// TIA Portal project "s14_code" (V21)

(* hardware
DEVICE "S7-1500/ET200MP station_1"  S7-1500 station
   slot 0: "Rail_0"  Rack  6ES7 590-1***0-0AA0
   slot 1: "ZZPLC"  CPU 1511-1 PN  6ES7 511-1AK00-0AB0  V1.8
      slot 3: "CPU display_1"  6ES7591-1AA00-0AA0
      slot 32768: "PROFINET interface_1"  X1
         slot 32769: "Port_1"  X1 P1
         slot 32770: "Port_2"  X1 P2
*)

// ===== PLC "ZZPLC"  CPU 1511-1 PN =====
// protected blocks, not shown: "ZZSCL"

VAR_GLOBAL   // PLC tag table "Default tag table"
   "ZZALPHA" AT %M10.0 : Bool;
   "ZZB" AT %M10.1 : Bool;
   "ZZC" AT %M10.2 : Bool;
   "ZZOUT" AT %M11.0 : Bool;
   "ZZN1" AT %MW20 : Int;
   "ZZN2" AT %MW22 : Int;
   "ZZN3" AT %MW24 : Int;
END_VAR

DATA_BLOCK "ZZDATA"   // DB1
{ S7_Optimized_Access := 'TRUE' }
VERSION : 0.1
   VAR
      run : Bool;
      speed : Int;
   END_VAR
BEGIN
END_DATA_BLOCK

DATA_BLOCK "ZZFB_DB"   // DB3
{ S7_Optimized_Access := 'TRUE' }
VERSION : 0.1
// stored: InstanceOfName ZZFB
"ZZFB"
BEGIN
END_DATA_BLOCK

DATA_BLOCK "ZZOUTER_DB"   // DB4
{ S7_Optimized_Access := 'TRUE' }
VERSION : 0.1
// stored: InstanceOfName ZZOUTER
"ZZOUTER"
BEGIN
END_DATA_BLOCK

DATA_BLOCK "ZZLAD2_DB"   // DB5
{ S7_Optimized_Access := 'TRUE' }
VERSION : 0.1
// stored: InstanceOfName ZZLAD2
"ZZLAD2"
BEGIN
END_DATA_BLOCK

// folder: System blocks/Program resources

DATA_BLOCK "IEC_Timer_0_DB"   // DB2
{ S7_Optimized_Access := 'TRUE' }
AUTHOR : Simatic
FAMILY : IEC
NAME : IEC_TMR
VERSION : 1.0
// stored: InstanceOfName IEC_TIMER
"IEC_TIMER"
BEGIN
END_DATA_BLOCK

// folder: (top level)

FUNCTION_BLOCK "ZZFB"   // FB1, LAD
{ S7_Optimized_Access := 'TRUE' }
VERSION : 0.1
   VAR_INPUT
      in1 : Bool;
   END_VAR
   VAR_OUTPUT
      out1 : Bool;
   END_VAR
   VAR_IN_OUT
      io1 : Int;
   END_VAR
BEGIN

REGION Network 1
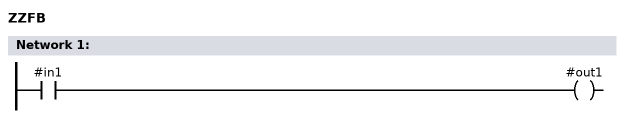
   RUNG wire#powerrail
      Contact( #in1 )
      Coil( #out1 )
   END_RUNG
   // the same network as SCL:
   #out1 := #in1;
END_REGION
END_FUNCTION_BLOCK

FUNCTION_BLOCK "ZZOUTER"   // FB2, LAD
{ S7_Optimized_Access := 'TRUE' }
VERSION : 0.1
   VAR
      inner : "ZZFB";
   END_VAR
BEGIN

REGION Network 1
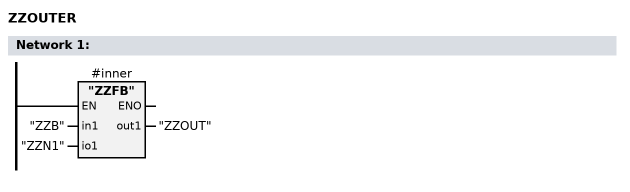
   RUNG wire#powerrail
      #inner(in1 := "ZZB", io1 := "ZZN1", out1 => "ZZOUT")
   END_RUNG
   // the same network as SCL:
   #inner(in1 := "ZZB", io1 := "ZZN1", out1 => "ZZOUT");   // "ZZFB"
END_REGION
END_FUNCTION_BLOCK

FUNCTION_BLOCK "ZZLAD2"   // FB3, LAD
{ S7_Optimized_Access := 'TRUE' }
VERSION : 0.1
   VAR
      memP : Bool;
      memN : Bool;
   END_VAR
   VAR RETAIN
      IEC_Counter_0_Instance : CTU_INT;
   END_VAR
   VAR
      IEC_Timer_0_Instance : TON_TIME;
   END_VAR
   VAR_TEMP   // added for the SCL form of the ladder/FBD networks
      _w1 : Bool;
   END_VAR
BEGIN

REGION Network 1
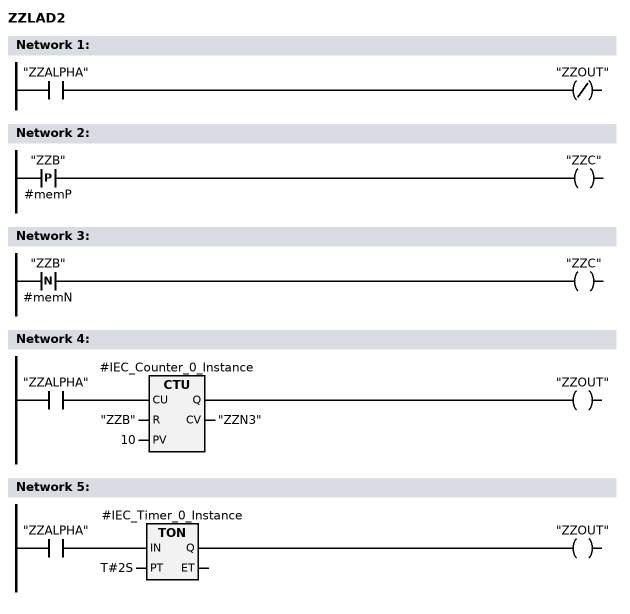
   RUNG wire#powerrail
      Contact( "ZZALPHA" )
      I_Coil( "ZZOUT" )
   END_RUNG
   // the same network as SCL:
   "ZZOUT" := NOT "ZZALPHA";
END_REGION

REGION Network 2
   RUNG wire#powerrail
      P_Contact(operand := "ZZB", bit := #memP)
      Coil( "ZZC" )
   END_RUNG
   // the same network as SCL:
   #_w1 := "ZZB" AND NOT #memP;   // rising edge of "ZZB"
   #memP := "ZZB";
   "ZZC" := #_w1;
END_REGION

REGION Network 3
   RUNG wire#powerrail
      N_Contact(operand := "ZZB", bit := #memN)
      Coil( "ZZC" )
   END_RUNG
   // the same network as SCL:
   #_w1 := NOT "ZZB" AND #memN;   // falling edge of "ZZB"
   #memN := "ZZB";
   "ZZC" := #_w1;
END_REGION

REGION Network 4
   #IEC_Counter_0_Instance(CU := "ZZALPHA", R := "ZZB", PV := 10, CV => "ZZN3");   // CTU
   "ZZOUT" := #IEC_Counter_0_Instance.Q;
END_REGION

REGION Network 5
   #IEC_Timer_0_Instance(IN := "ZZALPHA", PT := T#2S);   // TON
   "ZZOUT" := #IEC_Timer_0_Instance.Q;
END_REGION
END_FUNCTION_BLOCK

FUNCTION "ZZFBD" : Void   // FC1, FBD
{ S7_Optimized_Access := 'TRUE' }
VERSION : 0.1
BEGIN

REGION Network 1
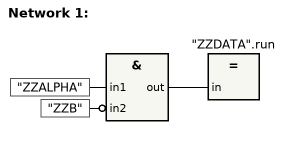
   "ZZDATA".run := "ZZALPHA" AND NOT "ZZB";
END_REGION
END_FUNCTION

FUNCTION "ZZSTL" : Void   // FC3, STL
{ S7_Optimized_Access := 'TRUE' }
VERSION : 0.1
BEGIN

REGION Network 1
         A     "ZZALPHA";
         AN    "ZZB";
         =     "ZZOUT";
END_REGION

REGION Network 2
         L     "ZZN1";
         L     5;
         +I;
         T     "ZZN3";
END_REGION
END_FUNCTION

FUNCTION "ZZSCL2" : Void   // FC4, SCL
{ S7_Optimized_Access := 'TRUE' }
VERSION : 0.1
BEGIN
   WHILE "ZZN1" < 10 DO
       "ZZN1" := "ZZN1" + 1;
   END_WHILE;
   REPEAT
       "ZZN2" := "ZZN2" + 1;
   UNTIL "ZZN2" > 5 END_REPEAT;
   CASE "ZZN3" OF
       1..5:
           "ZZOUT" := TRUE;
       6, 8:
           "ZZOUT" := FALSE;
       ELSE
           "ZZC" := TRUE;
   END_CASE;
   (/*multi-language comment*/)
END_FUNCTION

FUNCTION "ZZSTL2" : Void   // FC5, STL
{ S7_Optimized_Access := 'TRUE' }
VERSION : 0.1
BEGIN

REGION Network 1
   // line comment
         A     "ZZALPHA";  //inline comment
         JC    M001;
         L     1;
         T     "ZZN1";
   M001: NOP   0;
END_REGION

REGION Network 2
         CALL  "ZZFBD";
END_REGION

REGION Network 3
         CALL  "ZZFB", "ZZFB_DB"
         ( in1  := "ZZB",
           out1 := "ZZC",
           io1  := "ZZN2"
         );
END_REGION
END_FUNCTION

ORGANIZATION_BLOCK "Main"   // OB1, LAD, ProgramCycle
TITLE = "Main Program Sweep (Cycle)"
{ S7_Optimized_Access := 'TRUE' }
VERSION : 0.1
   VAR_INPUT
      Initial_Call : Bool;   // Initial call of this OB
      Remanence : Bool;   // =True, if remanent data are available
   END_VAR
   VAR_TEMP   // added for the SCL form of the ladder/FBD networks
      _w1 : Bool;
      _w2 : Bool;
   END_VAR
BEGIN

REGION Network 1: ZZ series
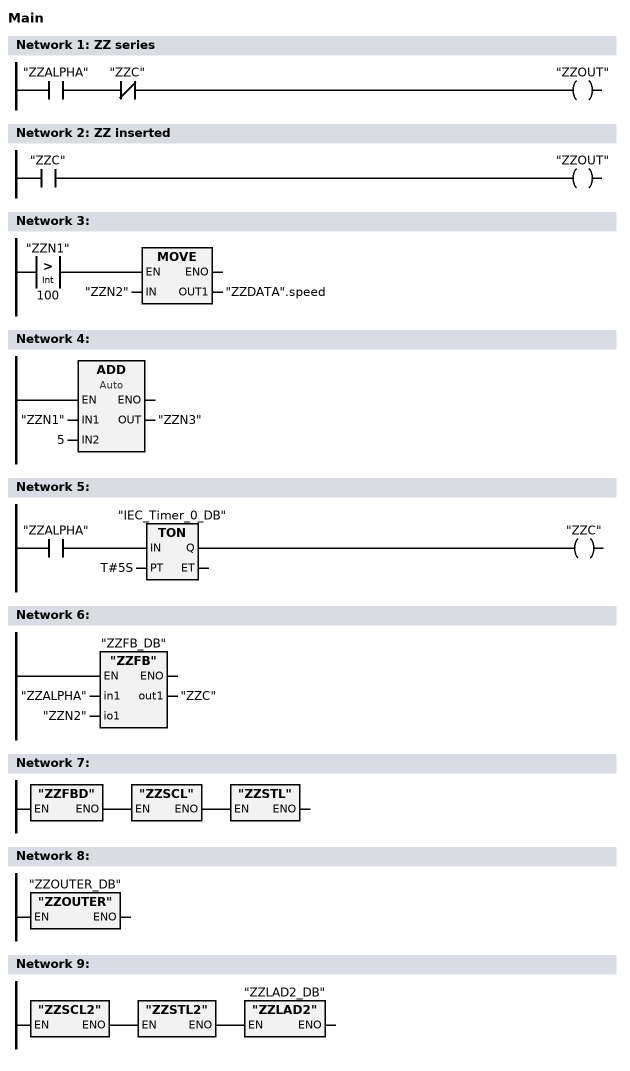
   RUNG wire#powerrail
      Contact( "ZZALPHA" )
      I_Contact( "ZZC" )
      Coil( "ZZOUT" )
   END_RUNG
   // the same network as SCL:
   "ZZOUT" := "ZZALPHA" AND NOT "ZZC";
END_REGION

REGION Network 2: ZZ inserted
   RUNG wire#powerrail
      Contact( "ZZC" )
      Coil( "ZZOUT" )
   END_RUNG
   // the same network as SCL:
   "ZZOUT" := "ZZC";
END_REGION

REGION Network 3
   RUNG wire#powerrail
      { S7_Templates := "SrcType := Int" } GT_Contact(in1 := "ZZN1", in2 := 100)
      Move(in := "ZZN2", out1 => "ZZDATA".speed)
   END_RUNG
   // the same network as SCL:
   IF "ZZN1" > 100 THEN "ZZDATA".speed := "ZZN2"; END_IF;
END_REGION

REGION Network 4
   RUNG wire#powerrail
      Add(in1 := "ZZN1", in2 := 5, out => "ZZN3")
   END_RUNG
   // the same network as SCL:
   "ZZN3" := "ZZN1" + 5;
END_REGION

REGION Network 5
   "IEC_Timer_0_DB".TON(IN := "ZZALPHA", PT := T#5S);
   "ZZC" := "IEC_Timer_0_DB".Q;
END_REGION

REGION Network 6
   RUNG wire#powerrail
      "ZZFB_DB"(in1 := "ZZALPHA", io1 := "ZZN2", out1 => "ZZC")
   END_RUNG
   // the same network as SCL:
   "ZZFB_DB"(in1 := "ZZALPHA", io1 := "ZZN2", out1 => "ZZC");   // "ZZFB"
END_REGION

REGION Network 7
   RUNG wire#powerrail
      "ZZFBD"()
      "ZZSCL"()
      "ZZSTL"()
   END_RUNG
   // the same network as SCL:
   "ZZFBD"(ENO => #_w1);
   "ZZSCL"(EN := #_w1, ENO => #_w2);
   IF #_w2 THEN "ZZSTL"(); END_IF;
END_REGION

REGION Network 8
   RUNG wire#powerrail
      "ZZOUTER_DB"()
   END_RUNG
   // the same network as SCL:
   "ZZOUTER_DB"();   // "ZZOUTER"
END_REGION

REGION Network 9
   RUNG wire#powerrail
      "ZZSCL2"()
      "ZZSTL2"()
      "ZZLAD2_DB"()
   END_RUNG
   // the same network as SCL:
   "ZZSCL2"(ENO => #_w1);
   "ZZSTL2"(EN := #_w1, ENO => #_w2);
   IF #_w2 THEN
       "ZZLAD2_DB"();   // "ZZLAD2"
   END_IF;
END_REGION
END_ORGANIZATION_BLOCK